TYPE T_Char : STrING(1); END_TYPE

(* stored: Version 1.1.0.1, ProductVersion 3.1.4024.14
   DUT T_Char: Id {e1d69649-c86c-0736-1a83-8c9a9b930ea3} *)
